FUNCTION_BLOCK FB_PIDR (* PID with Bumpless Transfer and Anti-Reset Windup, REAL PV+XOUT *)
  (* Standard: 61499-1-D.1 *)
  (* Version 0.0, 2004-09-06, JHC, Rockwell Automation *)
  (* Compiler header: package fb.rt.process; *)
  (* Compiler Java IBM VisualAge 3.0 *)
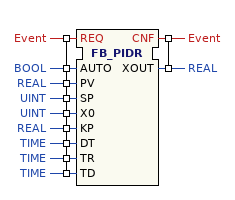
  EVENT_INPUT
    REQ WITH AUTO, PV, SP, X0, KP, TR, TD, DT;
  END_EVENT
  EVENT_OUTPUT
    CNF WITH XOUT;
  END_EVENT
  VAR_INPUT
    AUTO : BOOL; (* 0-manual,1-automatic *)
    PV : REAL; (* Process variable,0-100 percent *)
    SP : UINT; (* Set Point,0-100 percent *)
    X0 : UINT; (* Manual Output Setting,0-100 percent *)
    KP : REAL; (* Proportionality Constant *)
    DT : TIME := t#1s; (* Sampling Period *)
    TR : TIME; (* Reset Time *)
    TD : TIME; (* Derivative Time Constant *)
  END_VAR
  VAR_OUTPUT
    XOUT : REAL; (* Manipulated Variable,0-100 percent *)
  END_VAR
  VAR
    WASAUTO : BOOL;
    ERROR : REAL;
    ITERM : REAL;
    DTERM : REAL;
    X1 : REAL;
    X2 : REAL;
    X3 : REAL;
  END_VAR
  ALGORITHM REQ IN ST:
ERROR:=PV-SP;
IF AUTO THEN
  IF WASAUTO THEN
    ITERM:=ITERM+ERROR*DT/TR;
    DTERM:=(3*(PV-X3)+X1-X2)*TD/DT/10;
  ELSE
    ITERM:=(ERROR-X0)/KP;
    DTERM:=0;
  END_IF;
  XOUT:=-KP*ERROR-ITERM-DTERM;
ELSE XOUT:=X0;
END_IF
X3:=X2;X2:=X1;X1:=PV;
IF XOUT<0 THEN
  XOUT:=0;
  ITERM:=ITERM-ERROR*DT/TR;
ELSIF XOUT>100 THEN
  XOUT:=100;
  ITERM:=ITERM-ERROR*DT/TR;
END_IF;
WASAUTO:=AUTO;
CNF.serviceEvent(this);
  END_ALGORITHM
END_FUNCTION_BLOCK
